Fanuc KAREL source: ko00040.KL

PROGRAM KO00040
%STACKSIZE=65535
%PRIORITY=65535
%NOLOCKGROUP
VAR
P1 : POSITION
P2 : XYZWPR
F : BOOLEAN
OUT : JOINTPOS9
BEGIN
F=TRUE
-- UNSAFE_SOURCE_IR line 11: CALL_RESULT MIRROR(convert_position_to_xyzwprext(P1), convert_xyzwpr_to_position(P2), F)
END KO00040
